FUNCTION_BLOCK Test_StringSplitter_Handles_Empty_String EXTENDS TUnitTestBase
VAR
    StringSplitter : TStringSplitter;
END_VAR

Test_Started();

StringSplitter.Init(
    Str    := '',
    Delim1 := '$T',
    Delim2 := '');

Assertion.AssertEquals_STRING(
    Expected := '',
    Actual   := StringSplitter.GetNext(),
    ObjectName := _TestName,
    VariableName  := 'StringSplitter.GetNext()');

Assertion.AssertEquals_BOOL(
    Expected := FALSE,
    Actual   := StringSplitter.HasMore(),
    ObjectName := _TestName,
    VariableName  := 'StringSplitter.HasMore()');


Test_Finished();

END_FUNCTION_BLOCK

(* stored: Version 1.1.0.1, ProductVersion 3.1.4024.3
   POU Test_StringSplitter_Handles_Empty_String: Id {3a7cf2cc-79a9-0132-02fd-8eb652eaae4e}, SpecialFunc None *)
